TYPE DB_State :
(
	DB_Idle := -1,
	DB_Busy_Write,
	DB_Busy_Read,
	DB_Error
);
END_TYPE

(* stored: Version 1.1.0.1, ProductVersion 3.1.0.36
   DUT DB_State: Id {10f05811-40c5-4e6b-bd08-57c2c117ac8f} *)
